(* IEC 61131-3 sources: AXOpen/src/io/app/src, 2 files *)

(* ---- configuration.st ---- *)
USING AXOpen.Io;

CONFIGURATION MyConfiguration
    TASK Main(Interval := T#10ms, Priority := 1);
    PROGRAM P1 WITH Main: MyProgram;

    VAR_GLOBAL
        {S7.extern=ReadWrite}
        sandbox : SandboxContext;
        {S7.extern=ReadWrite}
        documentation : DocumentationContext;
        {S7.extern=ReadWrite}
        _rtc : AXOpen.S71500.Rtc;
        {S7.extern=ReadWrite}
        _rtm : AXOpen.S71500.Rtm;
        {S7.extern=ReadWrite}
        Inputs  AT %IB0 : Inputs;
        {S7.extern=ReadWrite}
		Outputs  AT %QB0 : Outputs;
        {S7.extern=ReadWrite}
        HwIDs : HwIDs;
    END_VAR

END_CONFIGURATION

(* ---- program.st ---- *)
USING AXOpen.Io;

PROGRAM MyProgram
    VAR_EXTERNAL
        sandbox : SandboxContext;
        documentation : DocumentationContext;
        _rtc : AXOpen.S71500.Rtc;
        _rtm : AXOpen.S71500.Rtm;
        Inputs : Inputs;
		Outputs : Outputs;
        // HwIDs : HwIDs;
    END_VAR

    VAR

    END_VAR

    VAR_TEMP

    END_VAR
    sandbox.InjectRtc(_rtc);
    sandbox.InjectRtm(_rtm);
    documentation.InjectRtc(_rtc);
    documentation.InjectRtm(_rtm);
    sandbox.Run();
    documentation.Run();
END_PROGRAM
